(* IEC 61131-3 sources: axopen.templates/axopen.template.simple/ax/templates-sources/unit/Data/Payloads, 2 files *)

(* ---- ProcessDataPayload.st ---- *)
NAMESPACE axosimple.UnitTemplate
    USING axosimple;
    USING AXOpen.Data;
    USING AXOpen.Core;
    USING System.Strings;

    {S7.extern=ReadWrite}
    CLASS ProcessDataPayload
        EXTENDS AXOpen.Data.AxoDataEntity
        VAR PUBLIC
            {#ix-set:AttributeName = "<#Unit header#>"}
            UnitHeader : UnitHeader;
        END_VAR
    END_CLASS
END_NAMESPACE

(* ---- TechnologyDataPayload.st ---- *)
NAMESPACE axosimple.UnitTemplate
    USING axosimple;
    USING AXOpen.Data;
    USING AXOpen.Core;
    USING System.Strings;

    {S7.extern=ReadWrite}
    CLASS TechnologyDataPayload
        EXTENDS AXOpen.Data.AxoDataEntity
        VAR PUBLIC
            Header : axosimple.TechnologyUnitHeader;
        END_VAR
    END_CLASS
END_NAMESPACE
